// TIA Portal project "3 Motor Senkronize Çalışma" (V18)

(* hardware
DEVICE "S7-1200 station_1"  S7-1200 Station
   slot 0: "Rack_0"  S7-1200 Rack  Rack  V1.0
   slot 1: "PLC_1"  CPU 1214C AC/DC/Rly  6ES7 214-1BG40-0XB0  V4.6
*)

// ===== PLC "PLC_1"  CPU 1214C AC/DC/Rly =====

VAR_GLOBAL   // PLC tag table "Default tag table"
   "Stop" AT %I0.0 : Bool;
   "Start" AT %I0.1 : Bool;
   "1. motor" AT %Q0.0 : Bool;
   "2. motor" AT %Q0.1 : Bool;
   "3. motor" AT %Q0.2 : Bool;
   "Tag_1" AT %M0.0 : Bool;
END_VAR

// folder: System blocks/Program resources

DATA_BLOCK "IEC_Timer_0_DB_1"   // DB2
{ S7_Optimized_Access := 'TRUE' }
AUTHOR : Simatic
FAMILY : IEC
NAME : IEC_TMR
VERSION : 1.0
// stored: InstanceOfName IEC_TIMER
"IEC_TIMER"
BEGIN
END_DATA_BLOCK

DATA_BLOCK "IEC_Timer_0_DB_3"   // DB4
{ S7_Optimized_Access := 'TRUE' }
AUTHOR : Simatic
FAMILY : IEC
NAME : IEC_TMR
VERSION : 1.0
// stored: InstanceOfName IEC_TIMER
"IEC_TIMER"
BEGIN
END_DATA_BLOCK

DATA_BLOCK "IEC_Timer_0_DB_4"   // DB5
{ S7_Optimized_Access := 'TRUE' }
AUTHOR : Simatic
FAMILY : IEC
NAME : IEC_TMR
VERSION : 1.0
// stored: InstanceOfName IEC_TIMER
"IEC_TIMER"
BEGIN
END_DATA_BLOCK

// folder: (top level)

ORGANIZATION_BLOCK "Main"   // OB1, LAD, ProgramCycle
TITLE = "Main Program Sweep (Cycle)"
{ S7_Optimized_Access := 'TRUE' }
VERSION : 0.1
// Senkronize Çalışma
   VAR_INPUT
      Initial_Call : Bool;   // Initial call of this OB
      Remanence : Bool;   // =True, if remanent data are available
   END_VAR
   VAR_TEMP   // added for the SCL form of the ladder/FBD networks
      _w1 : Bool;
   END_VAR
BEGIN

REGION Network 1
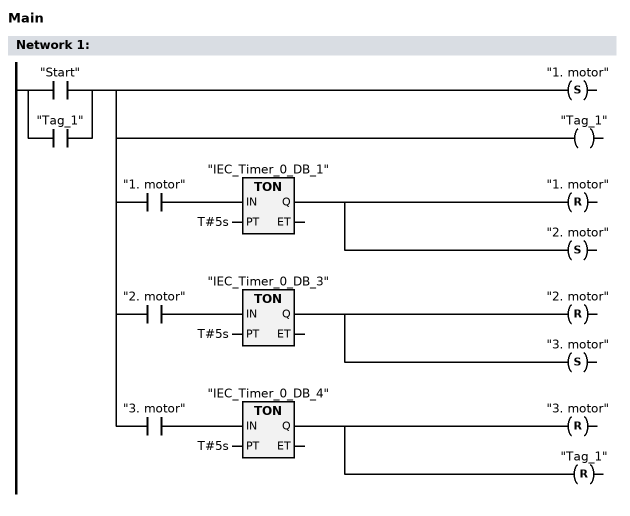
   #_w1 := "Start" OR "Tag_1";
   IF #_w1 THEN "1. motor" := TRUE; END_IF;
   "Tag_1" := #_w1;
   "IEC_Timer_0_DB_1".TON(IN := #_w1 AND "1. motor", PT := T#5s);
   IF "IEC_Timer_0_DB_1".Q THEN
       "1. motor" := FALSE;
       "2. motor" := TRUE;
   END_IF;
   "IEC_Timer_0_DB_3".TON(IN := #_w1 AND "2. motor", PT := T#5s);
   IF "IEC_Timer_0_DB_3".Q THEN
       "2. motor" := FALSE;
       "3. motor" := TRUE;
   END_IF;
   "IEC_Timer_0_DB_4".TON(IN := #_w1 AND "3. motor", PT := T#5s);
   IF "IEC_Timer_0_DB_4".Q THEN
       "3. motor" := FALSE;
       "Tag_1" := FALSE;
   END_IF;
END_REGION
END_ORGANIZATION_BLOCK